FUNCTION_BLOCK fb_debuger
VAR_INPUT
	in_flg_run: BOOL;
	in_flg_start: BOOL;
	in_var_cavQty: INT;
END_VAR
VAR_OUTPUT
	out_flg_gateLengthISSuccessed: BOOL;
	out_flg_dummySignal: BOOL;
	out_flg_lensSetDone: BOOL;
	out_flg_fiberSens: BOOL;
	out_flg_busy: BOOL;
	out_cav: INT;
END_VAR
VAR
	var_process: INT;
	var_cav: INT;
	delayTimer: TON;
END_VAR

IF in_flg_start AND in_flg_run THEN
	out_flg_busy := TRUE;
ELSE
	out_flg_busy := FALSE;
	var_process := 0;
	var_cav := gvl_param.var_productInfo[gvl_param.var_currentProductID].startCav - 1;
END_IF

CASE var_process OF
	0:
		out_flg_gateLengthISSuccessed := FALSE;
		out_flg_dummySignal := FALSE;
		out_flg_lensSetDone := FALSE;
		out_flg_fiberSens := FALSE;
		gvl_debug.cavConecctSkip := FALSE;
		delayTimer.IN := FALSE;
		IF out_flg_busy AND gvl_io.flg_requestLens THEN
			var_process := 1;
		END_IF
	1:
		gvl_debug.cavConecctSkip := TRUE;
		var_process := 2;
	2:
		//gate
		out_flg_gateLengthISSuccessed := TRUE;
		var_process := 3;
		
	3:
		//dummy signal
		IF gvl_debug.dummySignal THEN
			out_flg_dummySignal := TRUE;
			var_process := 4;
		ELSE
			var_process := 4;
		END_IF
	4:
		IF var_cav >= in_var_cavQty THEN
			var_cav := 1;
			out_cav := var_cav;
			var_process := 5;
		ELSE
			var_cav := var_cav + 1;
			out_cav := var_cav;
			var_process := 5;
		END_IF
	
	5:
		//lens set done
		delayTimer.IN := TRUE;
		out_flg_fiberSens := TRUE;
		IF delayTimer.Q THEN
			IF gvl_debug.flg_debug_run THEN
				out_flg_lensSetDone := TRUE;
				var_process := 0;
			END_IF
		END_IF
END_CASE
delayTimer(IN:= , PT:= T#3S , Q=> , ET=> );

END_FUNCTION_BLOCK

(* stored: Version 1.1.0.1, ProductVersion 3.1.4024.11
   POU fb_debuger: Id {45353351-3546-47d8-971e-515579eb02c1}, SpecialFunc None *)
